Yaskawa INFORM job: ROTINAS_ROBO.JBI

/JOB
//NAME ROTINAS_ROBO
///FOLDERNAME SERVICO
//POS
///NPOS 0,0,0,0,0,0
//INST
///DATE 2018/08/09 15:54
///ATTR SC,RW
NOP
''
IFTHENEXP IN#(2859)=ON OREXP IN#(2860)=ON
	 CALL JOB:DRESS
ENDIF
''
CALL JOB:TROCA_ELETRODO IF IN#(2860)=ON
END
